INTERFACE I_MoverPos

METHOD ChangeStep : BOOL
VAR_INPUT
	step : UDINT;
END_VAR
END_METHOD

PROPERTY ID : UDINT
GET
END_GET
END_PROPERTY

PROPERTY Position : LREAL
GET
END_GET
END_PROPERTY

METHOD SetData : BOOL
VAR_INPUT
	index : INT;
	value : LREAL;
END_VAR
END_METHOD

END_INTERFACE

(* stored: Version 1.1.0.1
   Itf I_MoverPos: Id {8759fd6a-e9a7-4f2f-bbfb-403f88fe374d}
   Method ChangeStep: Id {1bf0a4f5-16d9-48b8-96ca-459edb8a6339}
   Property ID: Id {a86fcca4-962b-4145-a7ff-2364534ed2ef}
   Get Get: Id {e6bf9d13-dca2-428b-9e80-46746d238a60}
   Property Position: Id {c8969d37-51d7-45ae-bf99-18c65816a161}
   Get Get: Id {4eb3f04f-2a30-4ac2-8609-0be88b06bbde}
   Method SetData: Id {456df2bd-33ec-4dae-90b0-1ac811984b35} *)
